FUNCTION_BLOCK JsonReader
VAR
	jsonParser : FB_JsonDomParser;
	jsonDocument : SJsonValue;
END_VAR
VAR CONSTANT
	INVALIDPARM : HRESULT := 16#9811070B;
	NOT_FOUND : HRESULT := 16#9811070C;
	INCOMPATIBLE : HRESULT := 16#9811070E;
END_VAR

METHOD PUBLIC LoadFromHttpRequest
VAR_INPUT
	HttpRequest : REFERENCE TO FB_IotHttpRequest;
END_VAR
jsonDocument := HttpRequest.GetJsonDomContent(jsonParser);
END_METHOD

METHOD PUBLIC LoadFromString
VAR_INPUT
	JsonString : T_MAXSTRING;
END_VAR
jsonDocument := jsonParser.ParseDocument(JsonString);
END_METHOD

METHOD PUBLIC ReadPath : HRESULT
VAR_INPUT
	Path : T_MaxString;
	Destination : ANY;
END_VAR
VAR
	result : HRESULT;
	jsonElement : I_JsonPathElement;
	jsonValue : SJsonValue;
	_BOOL : BOOL;
	_DINT : DINT;
	_LINT : LINT;
	_UDINT : UDINT;
	_ULINT : ULINT;
	_LREAL : LREAL;
	_STRING : POINTER TO STRING(1);
END_VAR
ParseJsonPath(Path,jsonElement);

IF FAILED(result) THEN
	ReadPath := result;
	RETURN;
END_IF

jsonValue := jsonElement.ResolveToSJsonValue(jsonParser,jsonDocument);
jsonElement.Dispose();

IF jsonValue = 0 THEN
	ReadPath := NOT_FOUND;
	RETURN;
END_IF

IF jsonParser.IsBool(jsonValue) THEN
	_BOOL := jsonParser.GetBool(jsonValue);
	ReadPath := Convert_BOOL_TO_(_BOOL,Destination);
	RETURN;
END_IF

IF jsonParser.IsInt(jsonValue) THEN
	_DINT := jsonParser.GetInt(jsonValue);
	ReadPath := Convert_DINT_TO_(_DINT,Destination);
	RETURN;
END_IF

IF jsonParser.IsInt64(jsonValue) THEN
	_LINT := jsonParser.GetInt64(jsonValue);
	ReadPath := Convert_LINT_TO_(_LINT,Destination);
	RETURN;
END_IF

IF jsonParser.IsUInt(jsonValue) THEN
	_UDINT := jsonParser.GetUInt(jsonValue);
	ReadPath := Convert_UDINT_TO_(_UDINT,Destination);
	RETURN;
END_IF

IF jsonParser.IsUInt64(jsonValue) THEN
	_ULINT := jsonParser.GetUInt64(jsonValue);
	ReadPath := Convert_ULINT_TO_(_ULINT,Destination);
	RETURN;
END_IF

IF jsonParser.IsDouble(jsonValue) THEN
	_LREAL := jsonParser.GetDouble(jsonValue);
	ReadPath := Convert_LREAL_TO_(_LREAL,Destination);
	RETURN;
END_IF

IF jsonParser.IsString(jsonValue) AND Destination.TypeClass = __SYSTEM.TYPE_CLASS.TYPE_STRING THEN
	_STRING := Destination.pValue;
	IF (jsonParser.CopyString(jsonValue,_STRING^,Destination.diSize) > 0) THEN;
		ReadPath := S_OK;
		RETURN;
	END_IF
END_IF
END_METHOD

END_FUNCTION_BLOCK

(* stored: Version 1.1.0.1, ProductVersion 3.1.4024.12
   POU JsonReader: Id {91fdfc05-0255-43a2-90ca-ffd8e5cfa080}, SpecialFunc None
   Method LoadFromHttpRequest: Id {db28d493-2bc0-424c-bb7e-318f6ef440be}
   Method LoadFromString: Id {b658e62e-3799-4095-9f1e-b3b4cdcb1654}
   Method ReadPath: Id {69ccef2a-b6a5-4daf-8700-f2215c7efe88} *)
